(* IEC 61131-3 sources: plc_generation_empirical_study/datasets/task_bank_v0_3/tasks/C08_B19_composite, 2 files *)

(* ---- interface.st ---- *)
FUNCTION_BLOCK C08_B19_composite
VAR_INPUT
    A_Start : BOOL;
    A_Stage1Done : BOOL;
    A_Stage2Done : BOOL;
    A_Stage3Done : BOOL;
    A_Pause : BOOL;
    A_Abort : BOOL;
    A_Reset : BOOL;
    B_ItemPresent : BOOL;
    B_RejectClass : BOOL;
    B_TransferDone : BOOL;
    B_Reset : BOOL;
    SubsystemBEnable : BOOL;
    CrossReset : BOOL;
END_VAR
VAR_OUTPUT
    A_Actuator1 : BOOL;
    A_Actuator2 : BOOL;
    A_Actuator3 : BOOL;
    A_Paused : BOOL;
    A_Complete : BOOL;
    A_Fault : BOOL;
    A_State : INT;
    B_Inspect : BOOL;
    B_AcceptGate : BOOL;
    B_RejectGate : BOOL;
    B_State : INT;
    CrossReady : BOOL;
    CrossBlocked : BOOL;
END_VAR
END_FUNCTION_BLOCK

(* ---- reference.st ---- *)
FUNCTION_BLOCK C08_B19_composite
VAR_INPUT
    A_Start : BOOL;
    A_Stage1Done : BOOL;
    A_Stage2Done : BOOL;
    A_Stage3Done : BOOL;
    A_Pause : BOOL;
    A_Abort : BOOL;
    A_Reset : BOOL;
    B_ItemPresent : BOOL;
    B_RejectClass : BOOL;
    B_TransferDone : BOOL;
    B_Reset : BOOL;
    SubsystemBEnable : BOOL;
    CrossReset : BOOL;
END_VAR
VAR_OUTPUT
    A_Actuator1 : BOOL;
    A_Actuator2 : BOOL;
    A_Actuator3 : BOOL;
    A_Paused : BOOL;
    A_Complete : BOOL;
    A_Fault : BOOL;
    A_State : INT;
    B_Inspect : BOOL;
    B_AcceptGate : BOOL;
    B_RejectGate : BOOL;
    B_State : INT;
    CrossReady : BOOL;
    CrossBlocked : BOOL;
END_VAR
VAR
    A_StageTimer : TON;
END_VAR

A_Complete := FALSE;
A_StageTimer(IN := (A_State > 0) AND (NOT A_Pause), PT := T#500ms);
IF A_Abort THEN
    A_State := 0;
    A_Fault := TRUE;
ELSIF A_StageTimer.Q THEN
    A_State := 0;
    A_Fault := TRUE;
ELSIF (A_State = 0) AND A_Reset AND (NOT A_Start) AND (NOT A_Abort) AND (NOT A_Stage1Done) AND (NOT A_Stage2Done) AND (NOT A_Stage3Done) THEN
    A_Fault := FALSE;
ELSIF NOT A_Fault THEN
    IF (A_State = 0) AND A_Start THEN
        A_State := 1;
    ELSIF NOT A_Pause THEN
        CASE A_State OF
            1: IF A_Stage1Done THEN A_State := 2; END_IF;
            2: IF A_Stage2Done THEN A_State := 3; END_IF;
            3: IF A_Stage3Done THEN A_State := 0; A_Complete := TRUE; END_IF;
            ELSE A_State := 0;
        END_CASE;
    END_IF;
END_IF;
A_Paused := (A_State > 0) AND A_Pause AND (NOT A_Fault);
A_Actuator1 := (A_State = 1) AND (NOT A_Pause) AND (NOT A_Fault);
A_Actuator2 := (A_State = 2) AND (NOT A_Pause) AND (NOT A_Fault);
A_Actuator3 := (A_State = 3) AND (NOT A_Pause) AND (NOT A_Fault);

IF CrossReset THEN
    CrossReady := FALSE;
ELSIF A_Actuator1 THEN
    CrossReady := TRUE;
END_IF;
CrossBlocked := SubsystemBEnable AND (NOT CrossReady);

IF SubsystemBEnable AND CrossReady THEN
    IF B_Reset THEN
        B_State := 0;
    ELSE
        CASE B_State OF
            0: IF B_ItemPresent THEN B_State := 1; END_IF;
            1: IF B_RejectClass THEN B_State := 3; ELSE B_State := 2; END_IF;
            2: IF B_TransferDone THEN B_State := 0; END_IF;
            3: IF B_TransferDone THEN B_State := 0; END_IF;
            ELSE B_State := 0;
        END_CASE;
    END_IF;
    B_Inspect := B_State = 1;
    B_AcceptGate := B_State = 2;
    B_RejectGate := B_State = 3;
ELSE
    B_Inspect := FALSE;
    B_AcceptGate := FALSE;
    B_RejectGate := FALSE;
    B_State := 0;
END_IF;

END_FUNCTION_BLOCK
